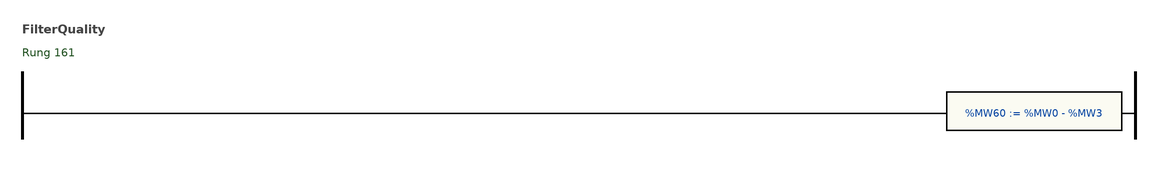
[picture p72: FilterQuality, ladder]

// Rung 161
  LD 1
  [ %MW60 := %MW0 - %MW3 ]
  // as ST:
  //   %MW60 := %MW0 - %MW3;
